{attribute 'qualified_only'}
VAR_GLOBAL
	FIOinputs : ARRAY[0..31, 0..7] OF BOOL;
	FIOoutputs : ARRAY [0..255] OF BOOL;
END_VAR

(* stored: Version 1.1.0.1
   GVL GVL_Factory_IO: Id {b6f2067d-5ef2-4457-bbc0-d96a38ed440a} *)
